// TwinCAT 3 PLC project PLC01
// ProgramVersion: 3.1.4024.0
// libraries:
//   Tc2_Standard, * (Beckhoff Automation GmbH)
//   Tc2_System, * (Beckhoff Automation GmbH)
//   Tc2_Utilities, * (Beckhoff Automation GmbH)
//   Tc3_Module, * (Beckhoff Automation GmbH)
//   VisuDialogs, * (System)
// project tree:
//   DUTs/ stRecordData.TcDUT
//   / GlobalTextList.TcGTLO, PlcTask.TcTTO, Visualization Manager.TcVMO (not stored)
//   GVLs/ GVL.TcGVL
//   POUs/ MAIN.TcPOU, prgFileRead.TcPOU, prgFileWrite.TcPOU
//   VISUs/ Footer.TcVIS, Reading.TcVIS, Writing.TcVIS
// real-time tasks:
//   TASK PlcTask: cycle T#10ms, priority 20, ADS port 350

CONFIGURATION PLC01
    RESOURCE PLC ON TwinCAT3
        TASK PlcTask(INTERVAL := T#10ms, PRIORITY := 20);
        PROGRAM MAIN WITH PlcTask : MAIN;
    END_RESOURCE
END_CONFIGURATION

// ---- DUTs/stRecordData.TcDUT
TYPE stRecordData :
STRUCT
	field01,field02,field03,field04,field05:T_MaxString;
END_STRUCT
END_TYPE

// ---- GVLs/GVL.TcGVL
{attribute 'qualified_only'}
VAR_GLOBAL
	data: ARRAY [1..MAX_CSV_ROWS] OF stRecordData := [(field01 := '1', field02 := '2', field03 := '3', field04 := '4', field05 := '5'), (field01 := '5', field02 := '4', field03 := '3', field04 := '2', field05 := '1'), 98(())];
	emptyData:stRecordData;
	recordFileNow, readFileNow: BOOL;
	readData:ARRAY[1..MAX_CSV_ROWS] OF stRecordData;
	sFileName: T_MaxString := 'C:/Relat/File.csv';
END_VAR
VAR_GLOBAL CONSTANT
	MAX_CSV_ROWS 			: UDINT := 100;
	MAX_CSV_COLUMNS 		: UDINT := 5;
	MAX_CSV_FIELD_LENGTH	: UDINT := 100;
END_VAR

// ---- POUs/MAIN.TcPOU
PROGRAM MAIN
VAR
END_VAR

prgFileWrite();
prgFileRead();

END_PROGRAM

// ---- POUs/prgFileWrite.TcPOU
PROGRAM prgFileWrite
VAR

	step: INT;
	bBusy: BOOL;
	bErr: BOOL;
	sErr: STRING;
	hFile: UINT;
	nRow: UDINT;
	nColumm: UDINT;
	
	fbFileOpen	: FB_FileOpen;(* Opens file *)
	fbFileClose	: FB_FileClose;(* Closes file *)
	fbFileWrite	: FB_FileWrite;(* Reads binary data *)
	fbWriter	: FB_CSVMemBufferWriter;(* Helper function block used to create CSV data bytes *)
	

	cbRecord:UDINT:=0;
	cbField: UDINT;
	field: ARRAY[0..GVL.MAX_CSV_FIELD_LENGTH] OF BYTE;
	record: ARRAY[0..1024] OF BYTE;
	iCycleCount: UDINT;
	iNumVezes:INT:=60;
	iVezAtual:INT;	
END_VAR

CASE step OF 
	0:
		IF GVL.recordFileNow THEN
			GVL.recordFileNow:=FALSE;
			bBusy:=TRUE;
			bErr:=FALSE;
			sErr:='';
			hFile:=0;
			nRow:=nColumm:=1;
			iCycleCount:=0;
			step:=10;
		END_IF
	10:
		//Nesse passo abrimos o arquivo em modo binário
		fbFileOpen(bExecute:= FALSE);
		fbFileOpen(sNetId:='' , sPathName:=GVL.sFileName , nMode:= FOPEN_MODEAPPEND OR FOPEN_MODEBINARY
			, ePath:= PATH_GENERIC, bExecute:= TRUE);
		step:=20;
	20:
		fbFileOpen(bExecute:=FALSE ,hFile=> hFile);
		IF NOT fbFileOpen.bBusy THEN
			IF NOT fbFileOpen.bError THEN
				step:=30;
			ELSE
				step:=100;
				sErr:='Error opening file';
				bErr:=TRUE;
			END_IF
		END_IF
	30:
		cbRecord:=0;
		fbWriter.eCmd:= eEnumCmd_First;
		IF nRow <=GVL.MAX_CSV_ROWS AND GVL.data[nRow].field01 <> '' THEN
			FOR nColumm:=1 TO GVL.MAX_CSV_COLUMNS BY 1 DO
				cbField:=0;
				CASE nColumm OF
					1:
						cbField:=ARG_TO_CSVFIELD(F_STRING(GVL.data[nRow].field01),TRUE,ADR(field),SIZEOF(field));
					2:
						cbField:=ARG_TO_CSVFIELD(F_STRING(GVL.data[nRow].field02),TRUE,ADR(field),SIZEOF(field));
					3:
						cbField:=ARG_TO_CSVFIELD(F_STRING(GVL.data[nRow].field03),TRUE,ADR(field),SIZEOF(field));
					4:
						cbField:=ARG_TO_CSVFIELD(F_STRING(GVL.data[nRow].field04),TRUE,ADR(field),SIZEOF(field));
					5:
						cbField:=ARG_TO_CSVFIELD(F_STRING(GVL.data[nRow].field05),TRUE,ADR(field),SIZEOF(field));
						
				END_CASE
				
				IF cbField > 0 THEN
					(* Add new field to the record buffer *)
					fbWriter( 	pBuffer := ADR( record ), cbBuffer := SIZEOF( record ), putValue :='',  pValue := ADR( field ), cbValue := cbField,
								bCRLF := ( nColumm = GVL.MAX_CSV_COLUMNS ) );(* bCRLF == TRUE => Write CRLF after the last field value *)
					IF fbWriter.bOk THEN
						fbWriter.eCmd 	:= eEnumCmd_Next;(* Write next field value *)
						cbRecord 		:= cbRecord + fbWriter.cbWrite;(* Calculate the new record size *)
					ELSE(* Error *)
						step := 100;
						RETURN;
					END_IF
				END_IF
				
			END_FOR
			nRow:=nRow+1;
			step:=40;
		ELSE
			step:=60;
		END_IF
	40:
		fbFileWrite( bExecute := FALSE );
		fbFileWrite( sNetId := '', hFile := hFile, pWriteBuff := ADR( record ), cbWriteLen := cbRecord, bExecute := TRUE );
		step := 50;		
	50:
		fbFileWrite( bExecute := FALSE, bError => bErr);
		IF NOT fbFileWrite.bBusy THEN
			IF NOT fbFileWrite.bError THEN
				step := 30;(* Write next record *)
			ELSE(* Error *)
				step := 100;
			END_IF
		END_IF
	60:
		fbFileClose( bExecute := FALSE );
		fbFileClose( sNetId := '', hFile := hFile, bExecute := TRUE );
		step := 70;	
	70:
		fbFileClose( bExecute := FALSE);
		IF ( NOT fbFileClose.bBusy ) THEN
			hFile := 0;
			step := 100;
		END_IF
	100:
		IF ( hFile <> 0 ) THEN
			step := 60; (* Close the source file *)
		ELSE
			bBusy := FALSE;
			step := 0;	(* Ready *)
			IF iVezAtual>=iNumVezes THEN
				iVezAtual:=0;
			END_IF
			iVezAtual:=iVezAtual+1;
		END_IF
END_CASE

END_PROGRAM

// ---- POUs/prgFileRead.TcPOU
PROGRAM prgFileRead
VAR
	sNetId			: T_AmsNetId := '';	(* TwinCAT system network address *)
	sCSVLine		: T_MaxString := '';(* Single CSV text line (row, record), we are using string as record buffer (your are able to see read fields)  *)
	sCSVField		: T_MaxString := '';(* Single CSV field value (column, record field) *)
	bBusy			: BOOL;
	bError			: BOOL;
	nErrId			: UDINT;
	nRow	 		: UDINT 	:= 0;(* Row number (record) *)
	nColumn			: UDINT 	:= 0;(* Column number (record field) *)
	hFile			: UINT		:= 0;(* File handle of the source file *)
	step			: DWORD 	:= 0;
	fbFileOpen		: FB_FileOpen;(* Opens file *)
	fbFileClose		: FB_FileClose;(* Closes file *)
	fbFileGets		: FB_FileGets;(* Reads one record (line) *)
	fbReader		: FB_CSVMemBufferReader;(* Helper function block used to parse CSV data bytes (single record line) *)

	i: UDINT;
	readTrig:R_TRIG;	
END_VAR

CASE step OF
	0:
		readTrig(CLK:=GVL.readFileNow);
		IF readTrig.Q THEN
			GVL.readFileNow 	:= FALSE;
			bBusy 	:= TRUE;
			bError	:= FALSE;
			nErrId	:= 0;
			hFile	:= 0;
			nRow	:= 1;
			nColumn	:= 0;
			step 		:= 1;
			FOR i:=1 TO GVL.MAX_CSV_ROWS DO
				GVL.readData[i]:=GVL.emptyData;
			END_FOR
		END_IF
	1:
		fbFileOpen(  bExecute := FALSE  );
		fbFileOpen( sNetId := sNetId, sPathName := GVL.sFileName, nMode := FOPEN_MODEREAD OR FOPEN_MODETEXT,(* Open file in TEXT mode! *)
					ePath := PATH_GENERIC, bExecute := TRUE );
		step := 2;
	2:
		fbFileOpen( bExecute := FALSE, bError => bError, nErrID => nErrID, hFile => hFile );
		IF NOT fbFileOpen.bBusy THEN
			IF NOT fbFileOpen.bError THEN
				step := 3;
			ELSE(* Error: file not found? *)
				step := 100;
			END_IF
		END_IF
	3:
		fbFileGets( bExecute := FALSE );
		fbFileGets( sNetId := sNetId, hFile := hFile, bExecute := TRUE );
		step := 4;
	4:
		fbFileGets( bExecute := FALSE, bError => bError, nErrID => nErrID, sLine => sCSVLine );
		IF NOT fbFileGets.bBusy THEN
			IF NOT fbFileGets.bError THEN
				IF fbFileGets.bEOF THEN
					step := 10;(* End of file reached => Close source file *)
				ELSE

					(* FB_FileGets returns text line without the CR (carriage return) character.
					We have to restore the CR character (replace the $L character with $R$L characters) *)
					IF RIGHT( sCSVLine, 1 ) = '$L' THEN
						sCSVLine := REPLACE( sCSVLine, '$R$L', 2, LEN(sCSVLine));
					END_IF

					step := 5;
				END_IF
			ELSE(* Error *)
				step := 100;
			END_IF
		END_IF
	5:
		fbReader.eCmd := eEnumCmd_First;(* Read first field value *)
		REPEAT
			fbReader( pBuffer := ADR( sCSVLine ), cbBuffer := SIZEOF( sCSVLine ), getValue => sCSVField );
			IF fbReader.bOk THEN
				fbReader.eCmd := eEnumCmd_Next;(* Read next field value *)

				CASE nColumn OF
					0:
						GVL.readData[nRow].field01:=  CSVFIELD_TO_STRING( sCSVField, FALSE );
					1:
						GVL.readData[nRow].field02:=  CSVFIELD_TO_STRING( sCSVField, FALSE );
					2:
						GVL.readData[nRow].field03:=  CSVFIELD_TO_STRING( sCSVField, FALSE );
					3:
						GVL.readData[nRow].field04:=  CSVFIELD_TO_STRING( sCSVField, FALSE );
					4:
						GVL.readData[nRow].field05:=  CSVFIELD_TO_STRING( sCSVField, FALSE );
				END_CASE

				nColumn := nColumn + 1;(* Increment number of read columns *)
				IF fbReader.bCRLF THEN(* CRLF == TRUE => End of reacord reached *)
					nRow 		:= nRow + 1;(* Increment number of read records *)
					nColumn 	:= 0;(* Reset number of columns *)
				END_IF

			ELSE(* Error: End of record reached or all fields read *)
				step := 3;(* Try to read next line *)
			END_IF
		UNTIL NOT fbReader.bOk
		END_REPEAT
	10:	(* Close source file *)
		fbFileClose( bExecute := FALSE );
		fbFileClose( sNetId := sNetId, hFile := hFile, bExecute := TRUE );
		step := 11;

	11:(* Wait until close not busy *)
		fbFileClose( bExecute := FALSE, bError => bError, nErrID => nErrID );
		IF ( NOT fbFileClose.bBusy ) THEN
			hFile := 0;
			step := 100;
		END_IF

	100: (* Error or ready step => cleanup *)
		IF ( hFile <> 0 ) THEN
			step := 10; (* Close the source file *)
		ELSE
			bBusy := FALSE;
			step := 0;	(* Ready *)
		END_IF	
END_CASE

END_PROGRAM

// ---- GlobalTextList.TcGTLO
TEXTLIST GlobalTextList
  846 = '%s'
  759 = 'Campo 01'
  911 = 'Campo 02'
  309 = 'Campo 03'
  171 = 'Campo 04'
  569 = 'Campo 05'
  739 = 'Escrita'
  289 = 'Field 01'
  136 = 'Field 02'
  593 = 'Field 03'
  40 = 'Field 04'
  389 = 'Field 05'
  344 = 'Filed 01'
  352 = 'Filed 02'
  4 = 'Filed 03'
  894 = 'Filed 04'
  700 = 'Filed 05'
  946 = 'Gravar'
  423 = 'Leitura'
  434 = 'Read'
  394 = 'Reading'
  736 = 'Write'
  247 = 'Writing'
END_TEXTLIST

// ---- VISUs/Footer.TcVIS
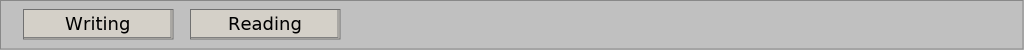
VISUALIZATION Footer  // 1024x50
    Button (23,9 150x30), "Writing"
        OnMouseClick: change screen: Writing
    Button (190,9 150x30), "Reading"
        OnMouseClick: change screen: Reading
END_VISUALIZATION

// ---- VISUs/Reading.TcVIS
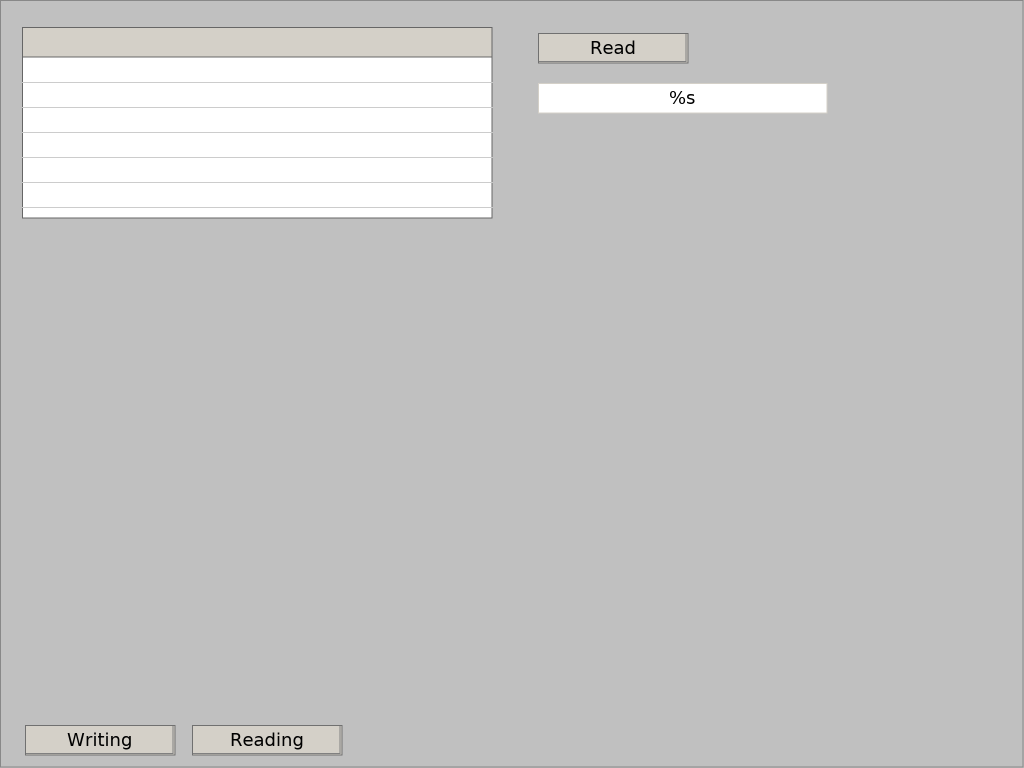
VISUALIZATION Reading  // 1024x768
    Table (22,27 470x191), data array: GVL.readData
        p3854506369: GVL.readData[INDEX].field01
        p1892666644: GVL.readData[INDEX].field02
        p338671338: GVL.readData[INDEX].field03
        p2170511999: GVL.readData[INDEX].field04
        p3723444502: GVL.readData[INDEX].field05
        p2232123230: Field 01
        p511219082: Field 02
        p1755163831: Field 03
        p4092479075: Field 04
        p2237128397: Field 05
    Button (538,33 150x30), "Read"
        tap GVL.readFileNow
    Textfield (538,83 289x30), "%s", text variable: GVL.sFileName
        OnMouseClick: write the text variable via Default
    Frame (2,716 1024x50)
        shows Footer()
END_VISUALIZATION

// ---- VISUs/Writing.TcVIS
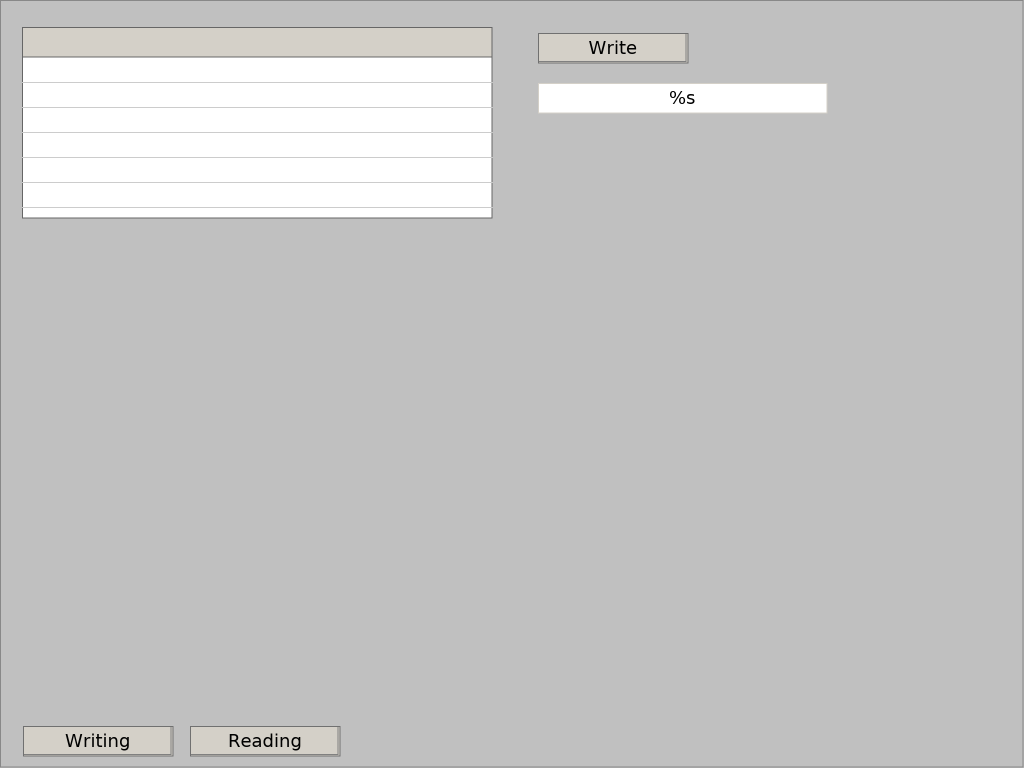
VISUALIZATION Writing  // 1024x768
    Table (22,27 470x191), data array: GVL.data
        p3854506369: GVL.data[INDEX].field01
        p1892666644: GVL.data[INDEX].field02
        p338671338: GVL.data[INDEX].field03
        p2170511999: GVL.data[INDEX].field04
        p3723444502: GVL.data[INDEX].field05
        p2232123230: Field 01
        p511219082: Field 02
        p1755163831: Field 03
        p4092479075: Field 04
        p2237128397: Field 05
    Button (538,33 150x30), "Write"
        tap GVL.recordFileNow
    Textfield (538,83 289x30), "%s", text variable: GVL.sFileName
        OnMouseClick: write the text variable via Default
    Frame (0,717 1024x50)
        shows Footer()
END_VISUALIZATION
